FUNCTION_BLOCK TcoMultiAxisPositionsRootContainer EXTENDS TcoCore.TcoObject
VAR_INPUT
END_VAR
VAR_OUTPUT
END_VAR
VAR
END_VAR

END_FUNCTION_BLOCK

(* stored: Version 1.1.0.1, ProductVersion 3.1.4024.12
   POU TcoMultiAxisPositionsRootContainer: Id {4a1b570d-6de6-03d7-1d34-24f1320276cd}, SpecialFunc None *)
